// TIA Portal V19 export
TYPE "LAF_typeDevDiagStateInstruct"
TITLE = State instructions / Anweisungen Status
// This data type contains the status information of the current instruction. / PN device Diagnose
// stored: Access Published
   STRUCT
      getName { ExternalAccessible := 'False'; ExternalVisible := 'False'; ExternalWritable := 'False'} : Bool;   // Get_Name
      geo2Log { ExternalAccessible := 'False'; ExternalVisible := 'False'; ExternalWritable := 'False'} : Bool;   // GEO2LOG
      moduleStates { ExternalAccessible := 'False'; ExternalVisible := 'False'; ExternalWritable := 'False'} : Bool;   // ModuleStates
      getDiag { ExternalAccessible := 'False'; ExternalVisible := 'False'; ExternalWritable := 'False'} : Bool;   // GET_DIAG
      getImData { ExternalAccessible := 'False'; ExternalVisible := 'False'; ExternalWritable := 'False'} : Bool;   // GET_IM_DATA
   END_STRUCT;
END_TYPE
